{attribute 'pack_mode' := '1'}
TYPE ST_RemoveTrafficLightDataIn :
STRUCT
	sCellID						: STRING(30);
	sID							: STRING(30);

END_STRUCT
END_TYPE

(* stored: Version 1.1.0.1, ProductVersion 3.1.4024.5
   DUT ST_RemoveTrafficLightDataIn: Id {9a14f0d8-10c0-4b42-8723-fce5aaa1eec6} *)
